{attribute "qualified_only"}
VAR_GLOBAL
	quotedFlag : BOOL;
END_VAR

(* stored: Version 1.1.0.1, ProductVersion 3.1.4026.18
   GVL GVL_Quoted: Id {00000000-0000-0000-0000-000000000011} *)
